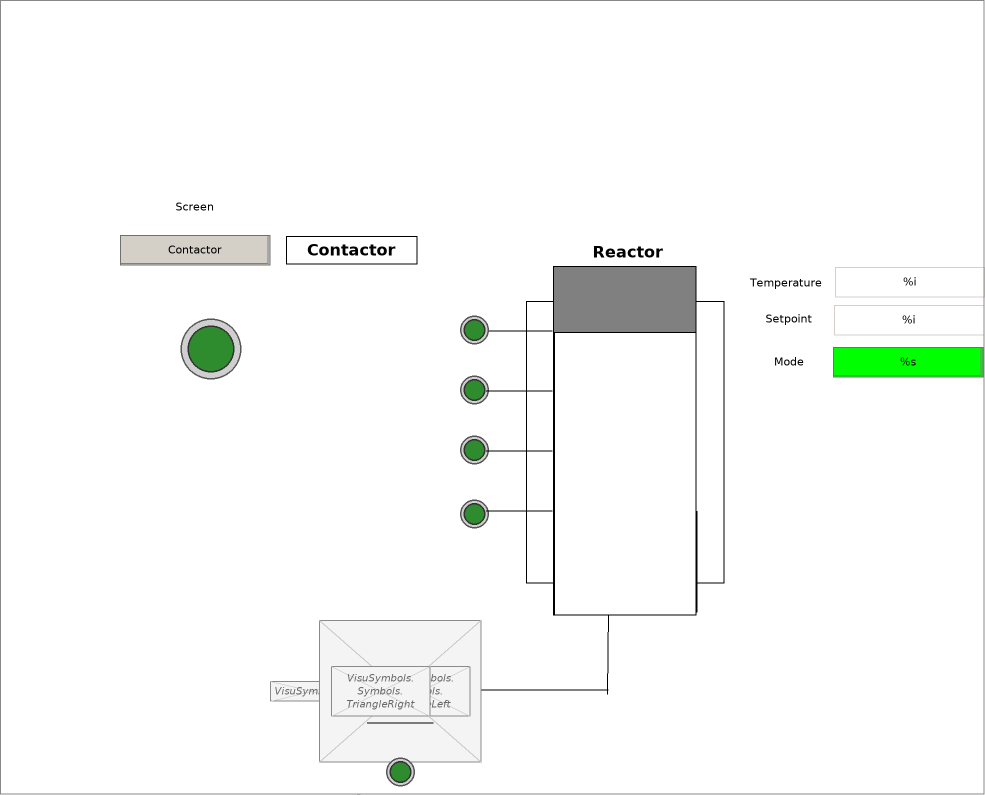
VISUALIZATION MainScreen  // 985x795
    Rectangle (526,301 198x282), colour toggle: HMI.bTemperatureControlSwitch
    RoundedRectangle (553,266 143x345)
    Label (120,192 150x30), "Screen"
    Button (120,235 150x30), "Contactor", colour toggle: HMI.bContactor
        toggle IO.bReactorTu
    Lamp1 (176,314 70x70), variable: IO.bReactorTu, style: Lamp-Lamp1-Green
    Line (552,331) (486,331)
    Lamp1 (458,311 33x38), variable: IO.bReactorHHy, style: Lamp-Lamp1-Green
    Lamp1 (458,371 33x38), variable: IO.bReactorHy, style: Lamp-Lamp1-Green
    Lamp1 (458,431 33x38), variable: IO.bReactorLy, style: Lamp-Lamp1-Green
    Lamp1 (458,495 33x38), variable: IO.bReactorLLy, style: Lamp-Lamp1-Green
    Textfield (834,305 150x30), "%i", text variable: HMI.iTemperatureSetpoint
        OnMouseDown: write the text variable via VisuDialogs.Numpad, min 40, max 120
    Label (715,261 142x44), "Temperature"
    Button (833,347 150x30), "%s", text variable: HMI.sTemperatureControlState, colour toggle: HMI.bTemperatureControlSwitch
        toggle HMI.bTemperatureControlSwitch
    Label (718,340 142x44), "Mode"
    Label (718,297 142x44), "Setpoint"
    Textfield (835,267 150x30), "%i", text variable: HMI.iTemperatureDisplayValue
    Line (608,611) (607,694)
    Line (608,690) (442,690)
    Line (552,391) (486,391)
    Line (552,451) (486,451)
    Line (552,511) (486,511)
    RoundedRectangle (286,236 131x28), "Contactor", invisible if: (NOT IO.bReactorTu) AND (NOT IO.bReactorHHy)
    RoundedRectangle (553,511 144x101), invisible if: (NOT IO.bReactorLLy) OR (IO.bReactorLy)
    Label (553,237 150x30), "Reactor"
    RoundedRectangle (553,452 143x162), invisible if: (NOT IO.bReactorLy) OR (IO.bReactorHy)
    RoundedRectangle (553,392 143x223), invisible if: (NOT IO.bReactorHy) OR (IO.bReactorHHy)
    RoundedRectangle (554,332 142x283), invisible if: (NOT IO.bReactorHHy)
    Image (270,681 83x20), image: VisuSymbols.Symbols.ArrowBoldLeft
    Image (319,620 162x142), invisible if: NOT IO.bReactorLu, image: ImagePool.VALVE
    Image (371,666 99x50), invisible if: IO.bReactorLu, image: VisuSymbols.Symbols.TriangleLeft
    Image (357,794 3x1), image: VisuSymbols.Symbols.TriangleRight
    Image (331,666 99x50), invisible if: IO.bReactorLu, image: VisuSymbols.Symbols.TriangleRight
    Line (433,723) (367,723)
    Lamp1 (384,753 33x38), variable: IO.bReactorLu, style: Lamp-Lamp1-Green
END_VISUALIZATION

(* stored: Version 1.1.0.1, ProductVersion 3.1.4024.9
   Visu MainScreen: Id {55a7e7e9-3ef6-43f8-8ba7-d69a5ee9abee} *)
